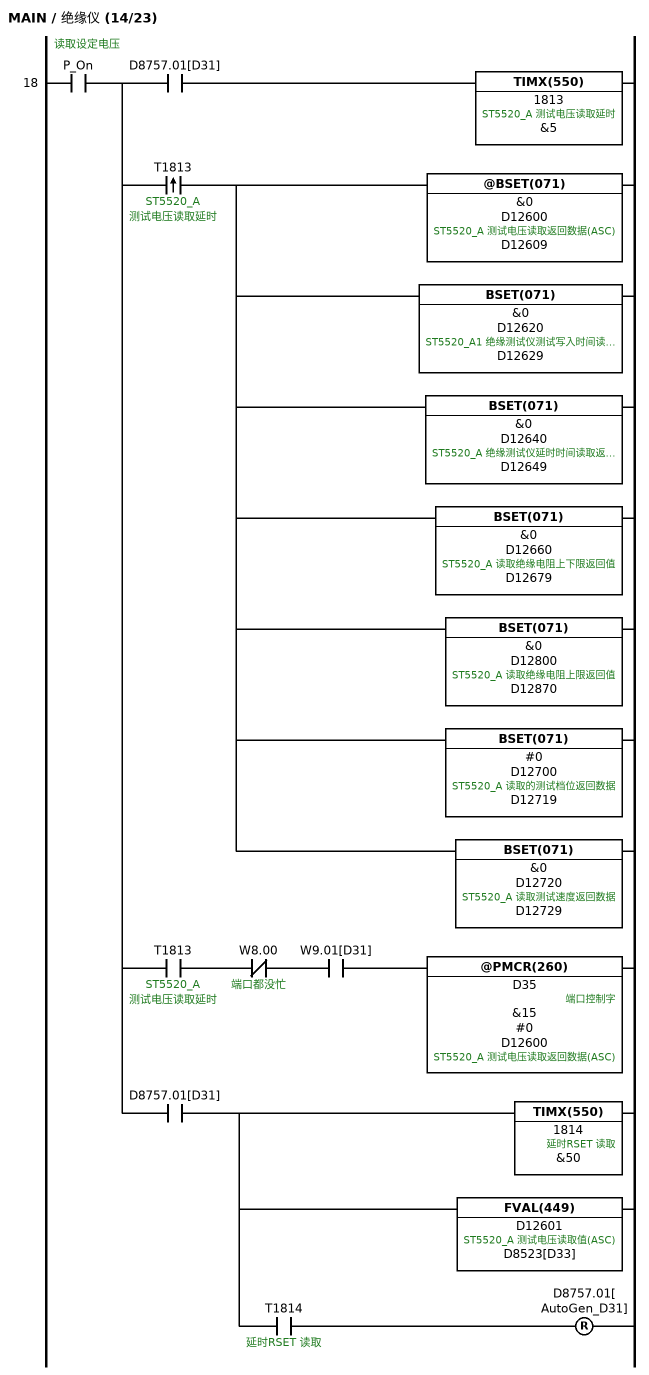
; [picture p48: MAIN / 绝缘仪, rungs 18-18]
; rung 18: 读取设定电压
LD P_On
OUT TR0
AND D8757.01[D31]
TIMX(550) 1813 &5  ; ST5520_A 测试电压读取延时
LD TR0
@AND T1813  ; ST5520_A 测试电压读取延时
@BSET(071) &0 D12600 D12609  ; ST5520_A 测试电压读取返回数据(ASC)
BSET(071) &0 D12620 D12629  ; ST5520_A1 绝缘测试仪测试写入时间读取值(ASC)
BSET(071) &0 D12640 D12649  ; ST5520_A 绝缘测试仪延时时间读取返回数据(ASC)
BSET(071) &0 D12660 D12679  ; ST5520_A 读取绝缘电阻上下限返回值
BSET(071) &0 D12800 D12870  ; ST5520_A 读取绝缘电阻上限返回值
BSET(071) #0 D12700 D12719  ; ST5520_A 读取的测试档位返回数据
BSET(071) &0 D12720 D12729  ; ST5520_A 读取测试速度返回数据
LD TR0
AND T1813  ; ST5520_A 测试电压读取延时
ANDNOT W8.00  ; 端口都没忙
AND W9.01[D31]
@PMCR(260) D35 &15 #0 D12600  ; 端口控制字, ST5520_A 测试电压读取返回数据(ASC)
LD TR0
AND D8757.01[D31]
TIMX(550) 1814 &50  ; 延时RSET 读取
FVAL(449) D12601 D8523[D33]  ; ST5520_A 测试电压读取值(ASC)
AND T1814  ; 延时RSET 读取
RSET D8757.01[AutoGen_D31]

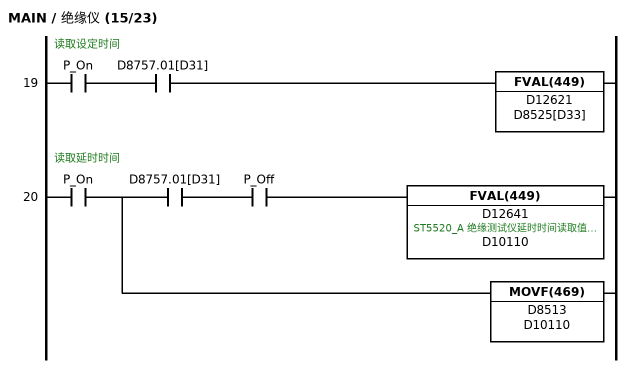
; rung 19: 读取设定时间
LD P_On
AND D8757.01[D31]
FVAL(449) D12621 D8525[D33]
; rung 20: 读取延时时间
LD P_On
OUT TR0
AND D8757.01[D31]
AND P_Off
FVAL(449) D12641 D10110  ; ST5520_A 绝缘测试仪延时时间读取值(ASC)
LD TR0
MOVF(469) D8513 D10110

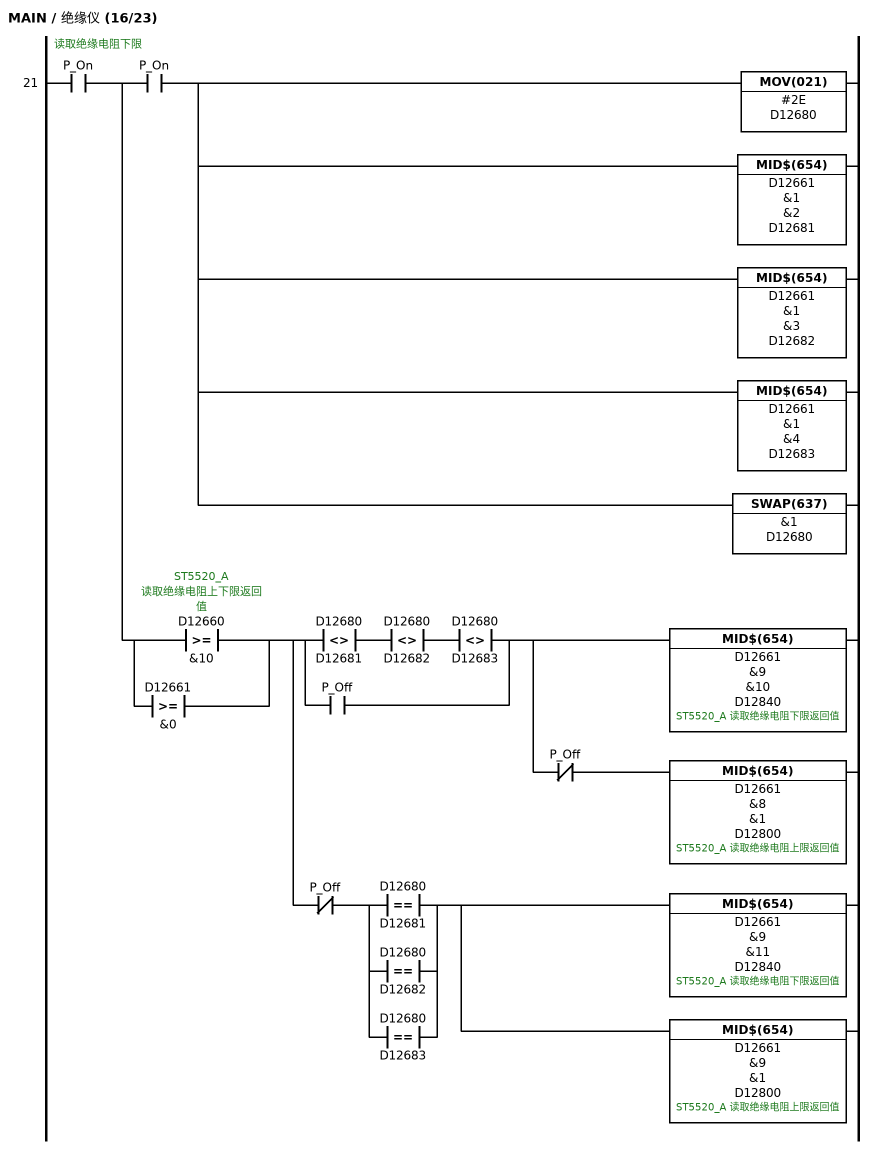
; rung 21: 读取绝缘电阻下限
LD P_On
OUT TR0
AND P_On
MOV(021) #2E D12680
MID$(654) D12661 &1 &2 D12681
MID$(654) D12661 &1 &3 D12682
MID$(654) D12661 &1 &4 D12683
SWAP(637) &1 D12680
LD TR0
LD>=(325) D12660 &10  ; ST5520_A 读取绝缘电阻上下限返回值
OR>=(325) D12661 &0
ANDLD
OUT TR0
LD<>(305) D12680 D12681
AND<>(305) D12680 D12682
AND<>(305) D12680 D12683
OR P_Off
ANDLD
MID$(654) D12661 &9 &10 D12840  ; ST5520_A 读取绝缘电阻下限返回值
ANDNOT P_Off
MID$(654) D12661 &8 &1 D12800  ; ST5520_A 读取绝缘电阻上限返回值
LD TR0
ANDNOT P_Off
LD=(300) D12680 D12681
OR=(300) D12680 D12682
OR=(300) D12680 D12683
ANDLD
MID$(654) D12661 &9 &11 D12840  ; ST5520_A 读取绝缘电阻下限返回值
MID$(654) D12661 &9 &1 D12800  ; ST5520_A 读取绝缘电阻上限返回值

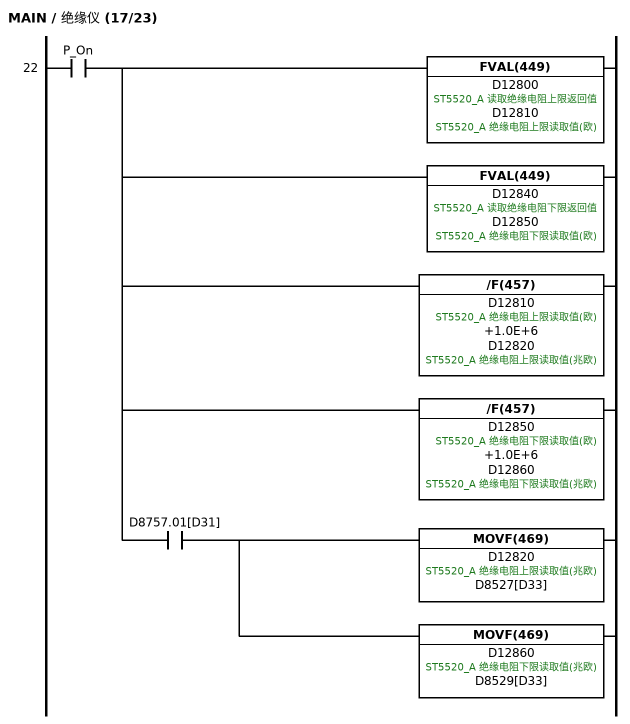
; rung 22
LD P_On
FVAL(449) D12800 D12810  ; ST5520_A 读取绝缘电阻上限返回值, ST5520_A 绝缘电阻上限读取值(欧)
FVAL(449) D12840 D12850  ; ST5520_A 读取绝缘电阻下限返回值, ST5520_A 绝缘电阻下限读取值(欧)
/F(457) D12810 +1.0E+6 D12820  ; ST5520_A 绝缘电阻上限读取值(欧), ST5520_A 绝缘电阻上限读取值(兆欧)
/F(457) D12850 +1.0E+6 D12860  ; ST5520_A 绝缘电阻下限读取值(欧), ST5520_A 绝缘电阻下限读取值(兆欧)
AND D8757.01[D31]
MOVF(469) D12820 D8527[D33]  ; ST5520_A 绝缘电阻上限读取值(兆欧)
MOVF(469) D12860 D8529[D33]  ; ST5520_A 绝缘电阻下限读取值(兆欧)

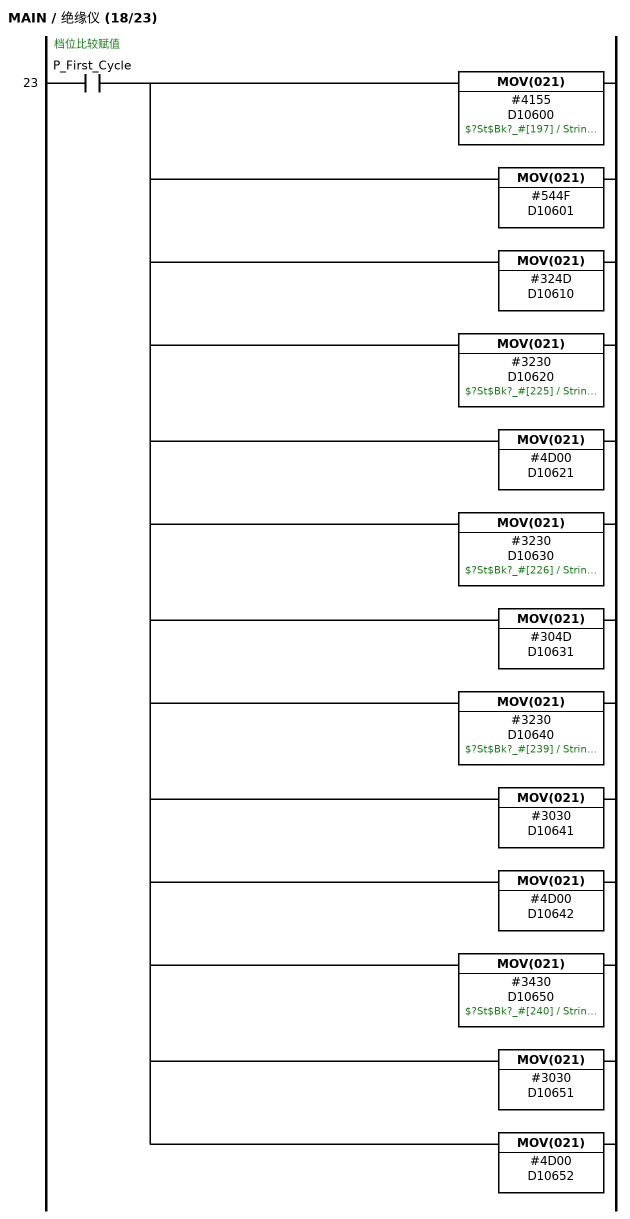
; rung 23: 档位比较赋值
LD P_First_Cycle
MOV(021) #4155 D10600  ; $?St$Bk?_#[197] / String "AUTO"$?St$Bk?_#[197]
MOV(021) #544F D10601
MOV(021) #324D D10610
MOV(021) #3230 D10620  ; $?St$Bk?_#[225] / String "20M"$?St$Bk?_#[225]
MOV(021) #4D00 D10621
MOV(021) #3230 D10630  ; $?St$Bk?_#[226] / String "200M"$?St$Bk?_#[226]
MOV(021) #304D D10631
MOV(021) #3230 D10640  ; $?St$Bk?_#[239] / String "2000M"$?St$Bk?_#[239]
MOV(021) #3030 D10641
MOV(021) #4D00 D10642
MOV(021) #3430 D10650  ; $?St$Bk?_#[240] / String "4000M"$?St$Bk?_#[240]
MOV(021) #3030 D10651
MOV(021) #4D00 D10652

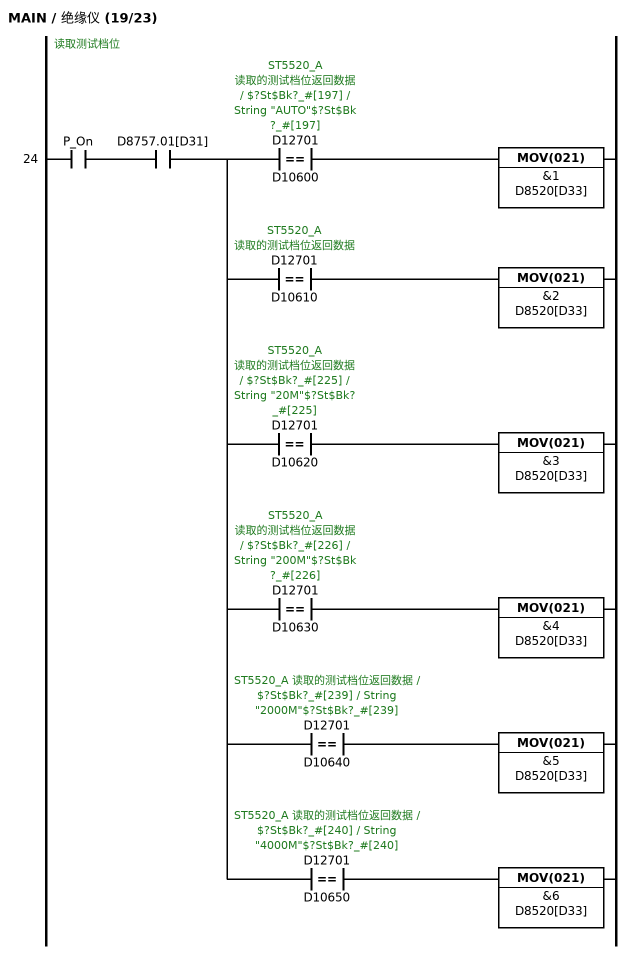
; rung 24: 读取测试档位
LD P_On
AND D8757.01[D31]
OUT TR0
AND=$(670) D12701 D10600  ; ST5520_A 读取的测试档位返回数据, $?St$Bk?_#[197] / String "AUTO"$?St$Bk?_#[197]
MOV(021) &1 D8520[D33]
LD TR0
AND=$(670) D12701 D10610  ; ST5520_A 读取的测试档位返回数据
MOV(021) &2 D8520[D33]
LD TR0
AND=$(670) D12701 D10620  ; ST5520_A 读取的测试档位返回数据, $?St$Bk?_#[225] / String "20M"$?St$Bk?_#[225]
MOV(021) &3 D8520[D33]
LD TR0
AND=$(670) D12701 D10630  ; ST5520_A 读取的测试档位返回数据, $?St$Bk?_#[226] / String "200M"$?St$Bk?_#[226]
MOV(021) &4 D8520[D33]
LD TR0
AND=$(670) D12701 D10640  ; ST5520_A 读取的测试档位返回数据, $?St$Bk?_#[239] / String "2000M"$?St$Bk?_#[239]
MOV(021) &5 D8520[D33]
LD TR0
AND=$(670) D12701 D10650  ; ST5520_A 读取的测试档位返回数据, $?St$Bk?_#[240] / String "4000M"$?St$Bk?_#[240]
MOV(021) &6 D8520[D33]

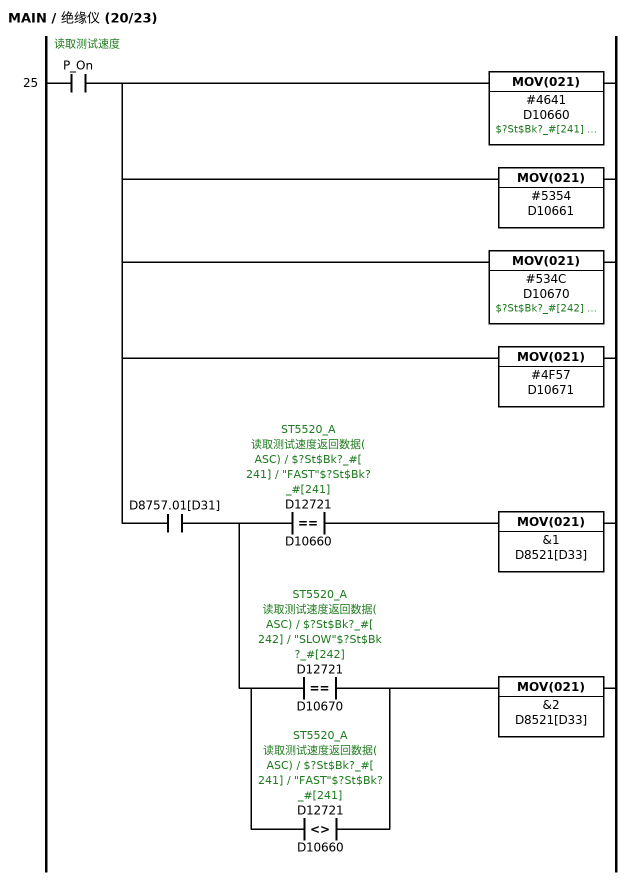
; rung 25: 读取测试速度
LD P_On
MOV(021) #4641 D10660  ; $?St$Bk?_#[241] / "FAST"$?St$Bk?_#[241]
MOV(021) #5354 D10661
MOV(021) #534C D10670  ; $?St$Bk?_#[242] / "SLOW"$?St$Bk?_#[242]
MOV(021) #4F57 D10671
AND D8757.01[D31]
OUT TR0
AND=$(670) D12721 D10660  ; ST5520_A 读取测试速度返回数据(ASC), $?St$Bk?_#[241] / "FAST"$?St$Bk?_#[241]
MOV(021) &1 D8521[D33]
LD TR0
LD=$(670) D12721 D10670  ; ST5520_A 读取测试速度返回数据(ASC), $?St$Bk?_#[242] / "SLOW"$?St$Bk?_#[242]
OR<>$(671) D12721 D10660  ; ST5520_A 读取测试速度返回数据(ASC), $?St$Bk?_#[241] / "FAST"$?St$Bk?_#[241]
ANDLD
MOV(021) &2 D8521[D33]

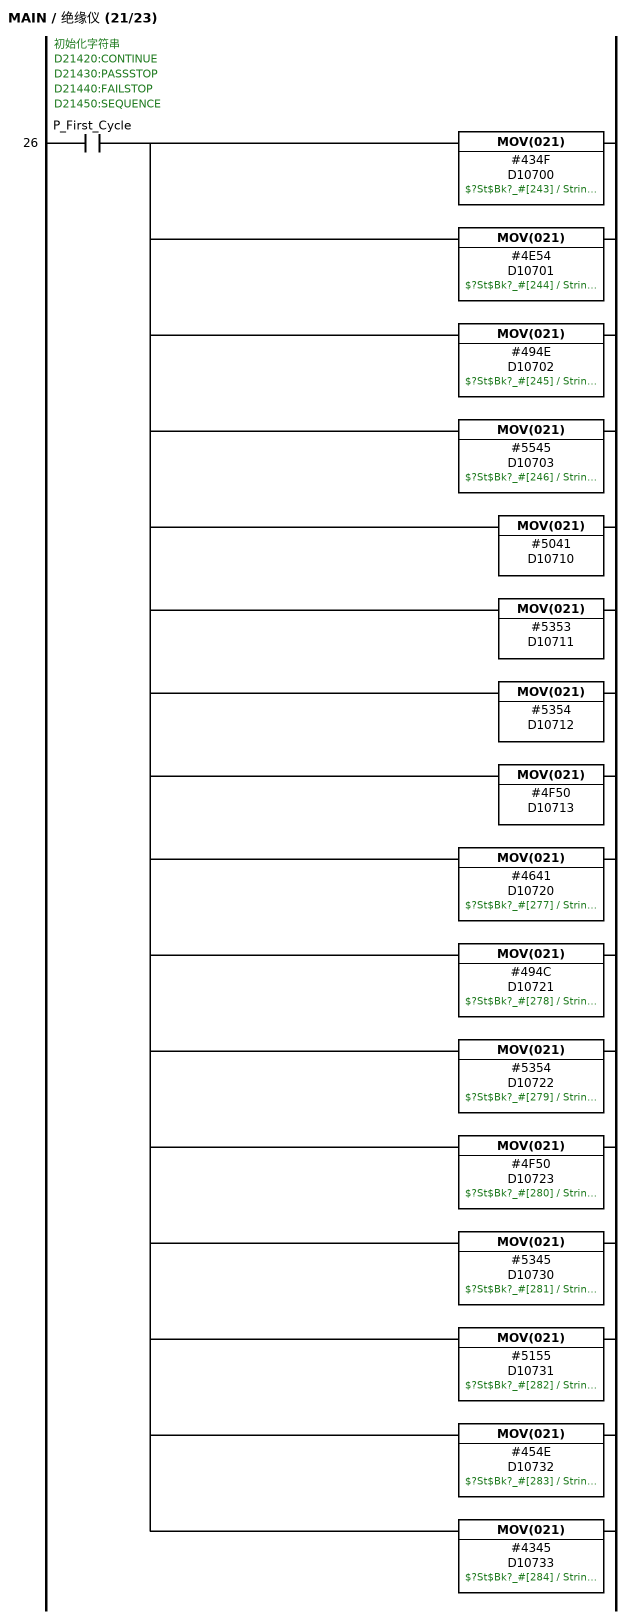
; rung 26: 初始化字符串 / D21420:CONTINUE / D21430:PASSSTOP / D21440:FAILSTOP / D21450:SEQUENCE
LD P_First_Cycle
MOV(021) #434F D10700  ; $?St$Bk?_#[243] / String "CONTINUE"$?St$Bk?_#[243]
MOV(021) #4E54 D10701  ; $?St$Bk?_#[244] / String "CONTINUE"$?St$Bk?_#[244]
MOV(021) #494E D10702  ; $?St$Bk?_#[245] / String "CONTINUE"$?St$Bk?_#[245]
MOV(021) #5545 D10703  ; $?St$Bk?_#[246] / String "CONTINUE"$?St$Bk?_#[246]
MOV(021) #5041 D10710
MOV(021) #5353 D10711
MOV(021) #5354 D10712
MOV(021) #4F50 D10713
MOV(021) #4641 D10720  ; $?St$Bk?_#[277] / String "FAILSTOP"$?St$Bk?_#[277]
MOV(021) #494C D10721  ; $?St$Bk?_#[278] / String "FAILSTOP"$?St$Bk?_#[278]
MOV(021) #5354 D10722  ; $?St$Bk?_#[279] / String "FAILSTOP"$?St$Bk?_#[279]
MOV(021) #4F50 D10723  ; $?St$Bk?_#[280] / String "FAILSTOP"$?St$Bk?_#[280]
MOV(021) #5345 D10730  ; $?St$Bk?_#[281] / String "SEQUENCE"$?St$Bk?_#[281]
MOV(021) #5155 D10731  ; $?St$Bk?_#[282] / String "SEQUENCE"$?St$Bk?_#[282]
MOV(021) #454E D10732  ; $?St$Bk?_#[283] / String "SEQUENCE"$?St$Bk?_#[283]
MOV(021) #4345 D10733  ; $?St$Bk?_#[284] / String "SEQUENCE"$?St$Bk?_#[284]

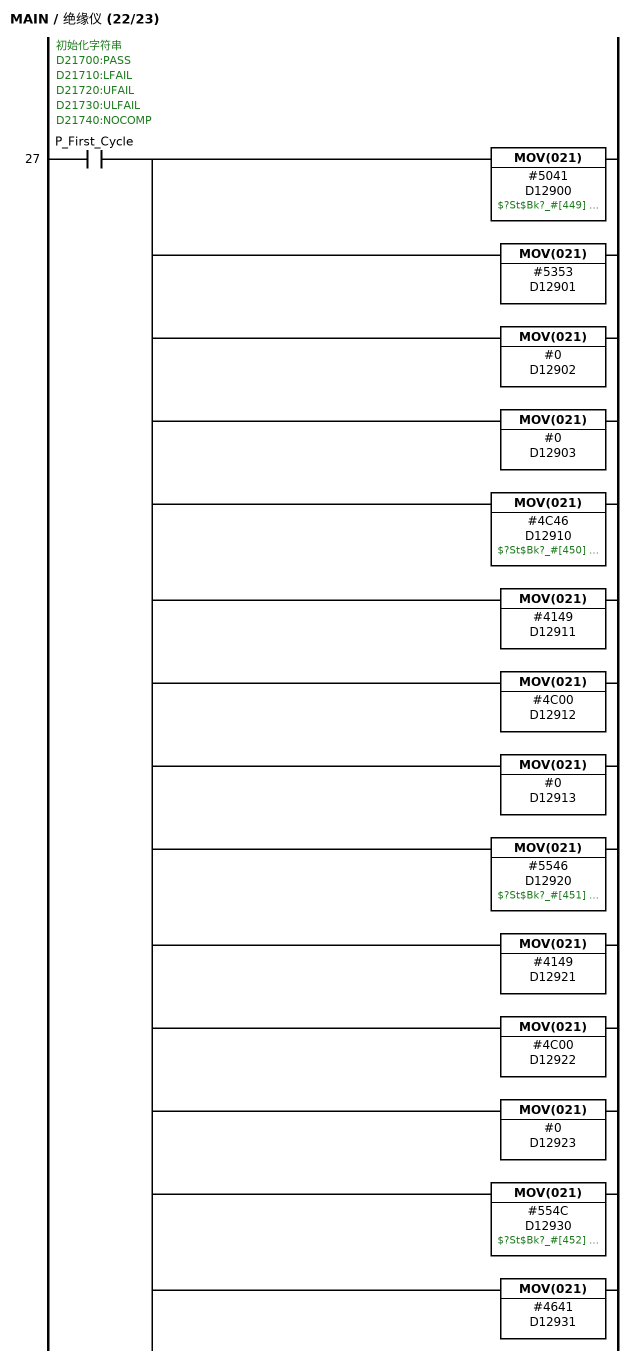

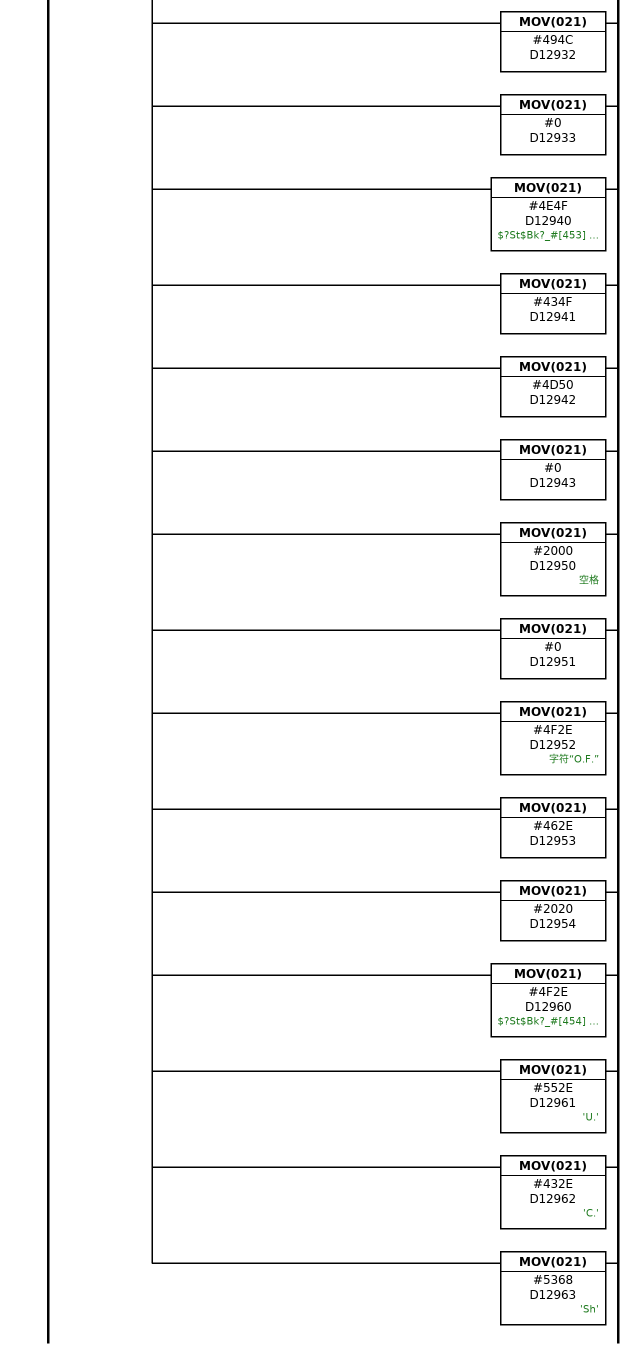
; rung 27: 初始化字符串 / D21700:PASS / D21710:LFAIL / D21720:UFAIL / D21730:ULFAIL / D21740:NOCOMP
LD P_First_Cycle
MOV(021) #5041 D12900  ; $?St$Bk?_#[449] / "PASS"$?St$Bk?_#[449]
MOV(021) #5353 D12901
MOV(021) #0 D12902
MOV(021) #0 D12903
MOV(021) #4C46 D12910  ; $?St$Bk?_#[450] / "LFAIL"$?St$Bk?_#[450]
MOV(021) #4149 D12911
MOV(021) #4C00 D12912
MOV(021) #0 D12913
MOV(021) #5546 D12920  ; $?St$Bk?_#[451] / "UFAIL"$?St$Bk?_#[451]
MOV(021) #4149 D12921
MOV(021) #4C00 D12922
MOV(021) #0 D12923
MOV(021) #554C D12930  ; $?St$Bk?_#[452] / "ULFAIL"$?St$Bk?_#[452]
MOV(021) #4641 D12931
MOV(021) #494C D12932
MOV(021) #0 D12933
MOV(021) #4E4F D12940  ; $?St$Bk?_#[453] / "NOCOMP"$?St$Bk?_#[453]
MOV(021) #434F D12941
MOV(021) #4D50 D12942
MOV(021) #0 D12943
MOV(021) #2000 D12950  ; 空格
MOV(021) #0 D12951
MOV(021) #4F2E D12952  ; 字符“O.F.”
MOV(021) #462E D12953
MOV(021) #2020 D12954
MOV(021) #4F2E D12960  ; $?St$Bk?_#[454] / "O."$?St$Bk?_#[454]
MOV(021) #552E D12961  ; 'U.'
MOV(021) #432E D12962  ; 'C.'
MOV(021) #5368 D12963  ; 'Sh'

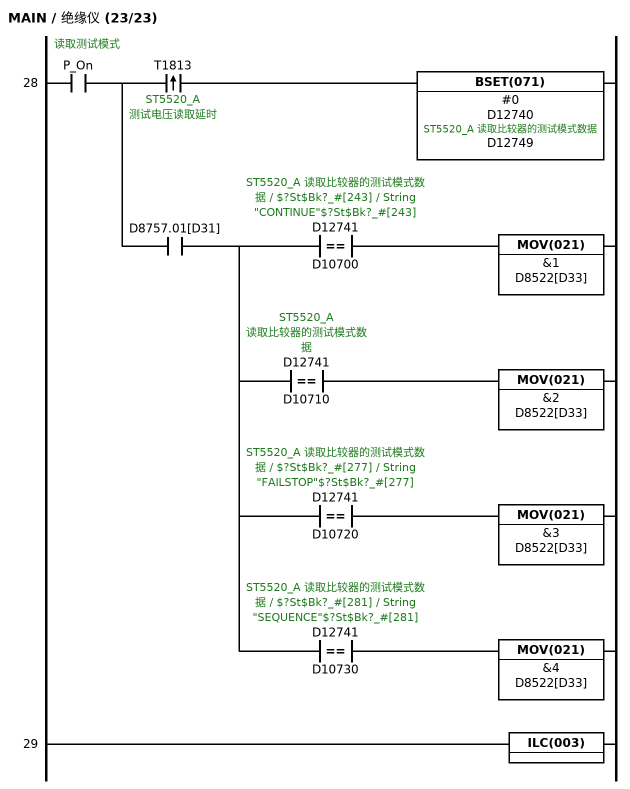
; rung 28: 读取测试模式
LD P_On
OUT TR0
@AND T1813  ; ST5520_A 测试电压读取延时
BSET(071) #0 D12740 D12749  ; ST5520_A 读取比较器的测试模式数据
LD TR0
AND D8757.01[D31]
OUT TR0
AND=$(670) D12741 D10700  ; ST5520_A 读取比较器的测试模式数据, $?St$Bk?_#[243] / String "CONTINUE"$?St$Bk?_#[243]
MOV(021) &1 D8522[D33]
LD TR0
AND=$(670) D12741 D10710  ; ST5520_A 读取比较器的测试模式数据
MOV(021) &2 D8522[D33]
LD TR0
AND=$(670) D12741 D10720  ; ST5520_A 读取比较器的测试模式数据, $?St$Bk?_#[277] / String "FAILSTOP"$?St$Bk?_#[277]
MOV(021) &3 D8522[D33]
LD TR0
AND=$(670) D12741 D10730  ; ST5520_A 读取比较器的测试模式数据, $?St$Bk?_#[281] / String "SEQUENCE"$?St$Bk?_#[281]
MOV(021) &4 D8522[D33]
; rung 29
ILC(003)

### Section 测试自动

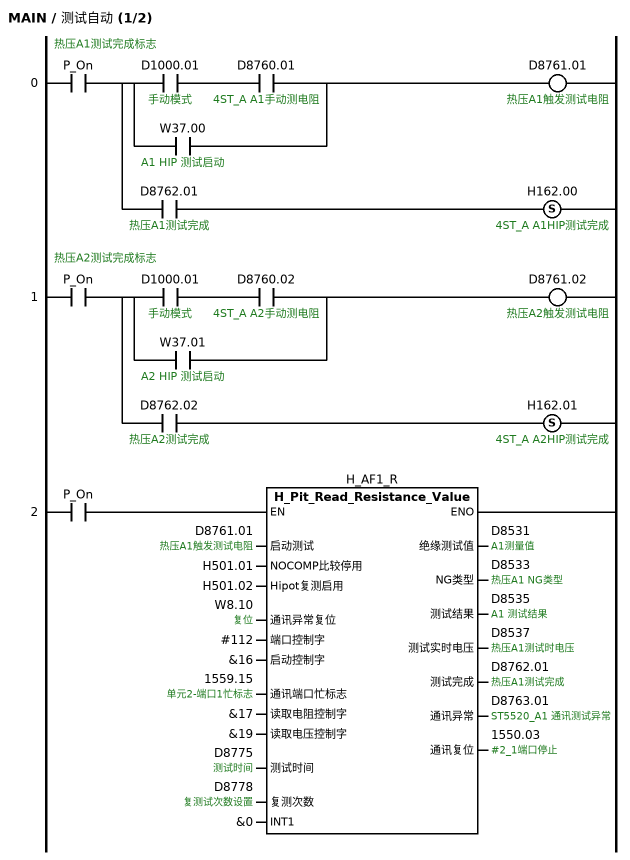
; rung 0: 热压A1测试完成标志
LD P_On
OUT TR0
LD D1000.01  ; 手动模式
AND D8760.01  ; 4ST_A A1手动测电阻
OR W37.00  ; A1 HIP 测试启动
ANDLD
OUT D8761.01  ; 热压A1触发测试电阻
LD TR0
AND D8762.01  ; 热压A1测试完成
SET H162.00  ; 4ST_A A1HIP测试完成
; rung 1: 热压A2测试完成标志
LD P_On
OUT TR0
LD D1000.01  ; 手动模式
AND D8760.02  ; 4ST_A A2手动测电阻
OR W37.01  ; A2 HIP 测试启动
ANDLD
OUT D8761.02  ; 热压A2触发测试电阻
LD TR0
AND D8762.02  ; 热压A2测试完成
SET H162.01  ; 4ST_A A2HIP测试完成
; rung 2
LD P_On
CALL H_AF1_R : H_Pit_Read_Resistance_Value (启动测试 := D8761.01, NOCOMP比较停用 := H501.01, Hipot复测启用 := H501.02, 通讯异常复位 := W8.10, 端口控制字 := #112, 启动控制字 := &16, 通讯端口忙标志 := 1559.15, 读取电阻控制字 := &17, 读取电压控制字 := &19, 测试时间 := D8775, 复测次数 := D8778, INT1 := &0, 绝缘测试值 => D8531, NG类型 => D8533, 测试结果 => D8535, 测试实时电压 => D8537, 测试完成 => D8762.01, 通讯异常 => D8763.01, 通讯复位 => 1550.03)  ; 热压A1触发测试电阻, 复位, 单元2-端口1忙标志, 测试时间, 复测试次数设置, A1测量值, 热压A1 NG类型, A1 测试结果, 热压A1测试时电压, 热压A1测试完成, ST5520_A1 通讯测试异常, #2_1端口停止

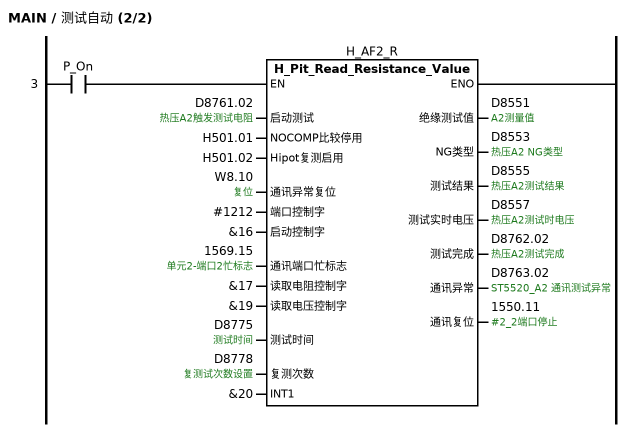
; rung 3
LD P_On
CALL H_AF2_R : H_Pit_Read_Resistance_Value (启动测试 := D8761.02, NOCOMP比较停用 := H501.01, Hipot复测启用 := H501.02, 通讯异常复位 := W8.10, 端口控制字 := #1212, 启动控制字 := &16, 通讯端口忙标志 := 1569.15, 读取电阻控制字 := &17, 读取电压控制字 := &19, 测试时间 := D8775, 复测次数 := D8778, INT1 := &20, 绝缘测试值 => D8551, NG类型 => D8553, 测试结果 => D8555, 测试实时电压 => D8557, 测试完成 => D8762.02, 通讯异常 => D8763.02, 通讯复位 => 1550.11)  ; 热压A2触发测试电阻, 复位, 单元2-端口2忙标志, 测试时间, 复测试次数设置, A2测量值, 热压A2 NG类型, 热压A2测试结果, 热压A2测试时电压, 热压A2测试完成, ST5520_A2 通讯测试异常, #2_2端口停止

### Section END
; rung 0
END(001)

## Program 进料定位 (cyclic task 1)

### Section Main

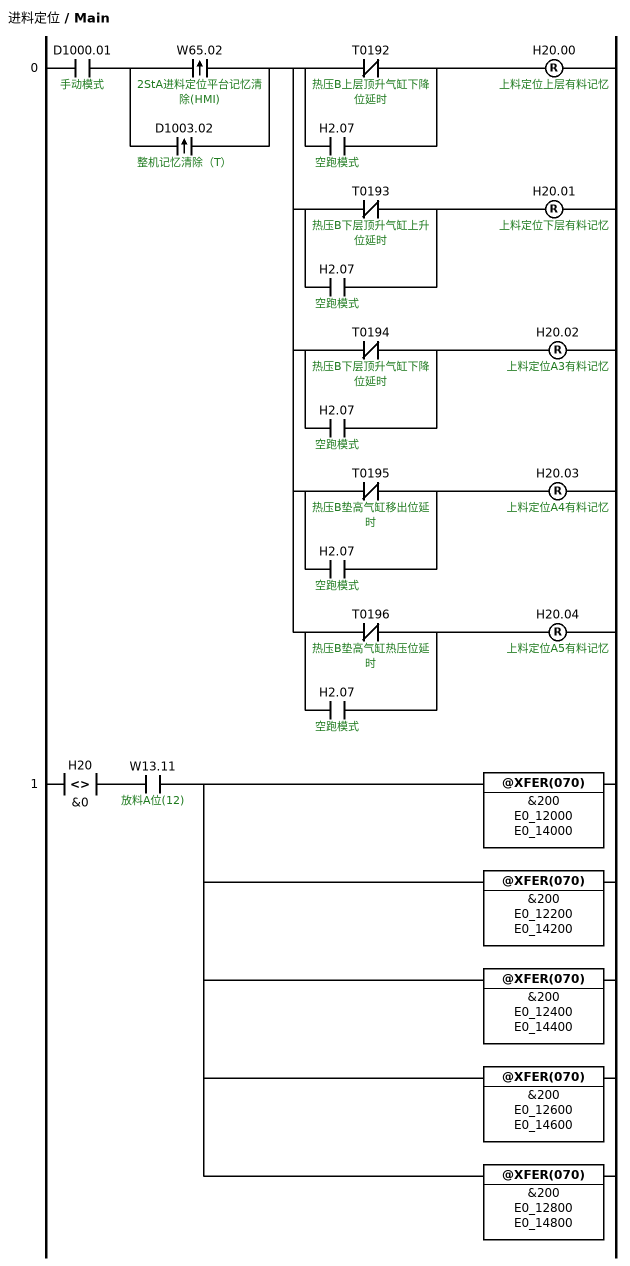
; rung 0
LD D1000.01  ; 手动模式
@LD W65.02  ; 2StA进料定位平台记忆清除(HMI)
@OR D1003.02  ; 整机记忆清除（T）
ANDLD
OUT TR0
LDNOT T0192  ; 热压B上层顶升气缸下降位延时
OR H2.07  ; 空跑模式
ANDLD
RSET H20.00  ; 上料定位上层有料记忆
LD TR0
LDNOT T0193  ; 热压B下层顶升气缸上升位延时
OR H2.07  ; 空跑模式
ANDLD
RSET H20.01  ; 上料定位下层有料记忆
LD TR0
LDNOT T0194  ; 热压B下层顶升气缸下降位延时
OR H2.07  ; 空跑模式
ANDLD
RSET H20.02  ; 上料定位A3有料记忆
LD TR0
LDNOT T0195  ; 热压B垫高气缸移出位延时
OR H2.07  ; 空跑模式
ANDLD
RSET H20.03  ; 上料定位A4有料记忆
LD TR0
LDNOT T0196  ; 热压B垫高气缸热压位延时
OR H2.07  ; 空跑模式
ANDLD
RSET H20.04  ; 上料定位A5有料记忆
; rung 1
LD<>(305) H20 &0
AND W13.11  ; 放料A位(12)
@XFER(070) &200 E0_12000 E0_14000
@XFER(070) &200 E0_12200 E0_14200
@XFER(070) &200 E0_12400 E0_14400
@XFER(070) &200 E0_12600 E0_14600
@XFER(070) &200 E0_12800 E0_14800

### Section _1ST进料定位

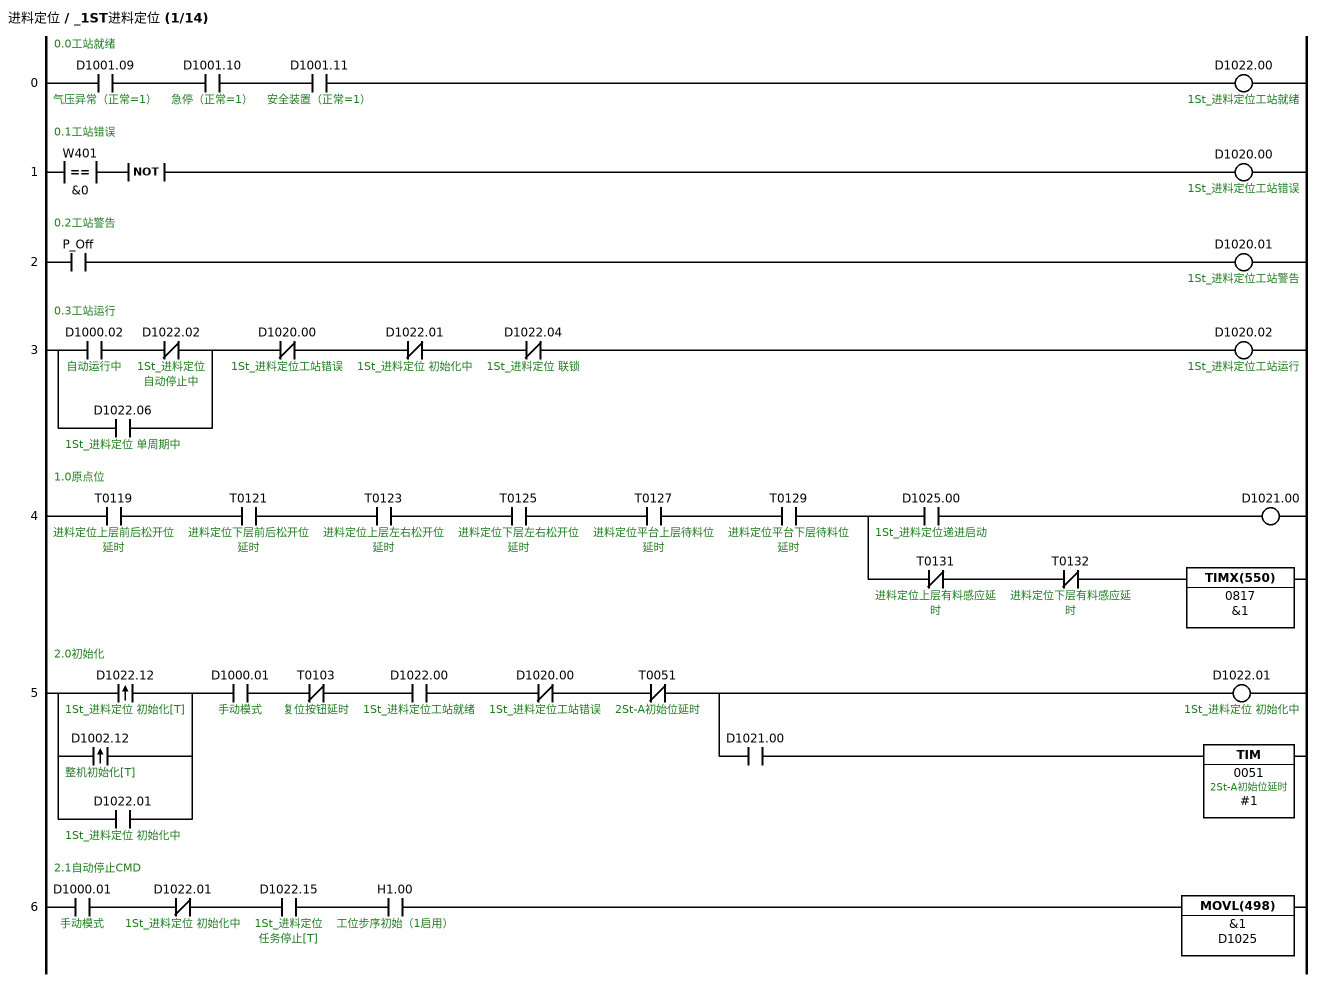
; rung 0: 0.0工站就绪
LD D1001.09  ; 气压异常（正常=1）
AND D1001.10  ; 急停（正常=1）
AND D1001.11  ; 安全装置（正常=1）
OUT D1022.00  ; 1St_进料定位工站就绪
; rung 1: 0.1工站错误
LD=(300) W401 &0
NOT(520)
OUT D1020.00  ; 1St_进料定位工站错误
; rung 2: 0.2工站警告
LD P_Off
OUT D1020.01  ; 1St_进料定位工站警告
; rung 3: 0.3工站运行
LD D1000.02  ; 自动运行中
ANDNOT D1022.02  ; 1St_进料定位 自动停止中
OR D1022.06  ; 1St_进料定位 单周期中
ANDNOT D1020.00  ; 1St_进料定位工站错误
ANDNOT D1022.01  ; 1St_进料定位 初始化中
ANDNOT D1022.04  ; 1St_进料定位 联锁
OUT D1020.02  ; 1St_进料定位工站运行
; rung 4: 1.0原点位
LD T0119  ; 进料定位上层前后松开位延时
AND T0121  ; 进料定位下层前后松开位延时
AND T0123  ; 进料定位上层左右松开位延时
AND T0125  ; 进料定位下层左右松开位延时
AND T0127  ; 进料定位平台上层待料位延时
AND T0129  ; 进料定位平台下层待料位延时
OUT TR0
AND D1025.00  ; 1St_进料定位递进启动
OUT D1021.00
LD TR0
ANDNOT T0131  ; 进料定位上层有料感应延时
ANDNOT T0132  ; 进料定位下层有料感应延时
TIMX(550) 0817 &1
; rung 5: 2.0初始化
@LD D1022.12  ; 1St_进料定位 初始化[T]
@OR D1002.12  ; 整机初始化[T]
OR D1022.01  ; 1St_进料定位 初始化中
AND D1000.01  ; 手动模式
ANDNOT T0103  ; 复位按钮延时
AND D1022.00  ; 1St_进料定位工站就绪
ANDNOT D1020.00  ; 1St_进料定位工站错误
ANDNOT T0051  ; 2St-A初始位延时
OUT D1022.01  ; 1St_进料定位 初始化中
AND D1021.00
TIM 0051 #1  ; 2St-A初始位延时
; rung 6: 2.1自动停止CMD
LD D1000.01  ; 手动模式
ANDNOT D1022.01  ; 1St_进料定位 初始化中
AND D1022.15  ; 1St_进料定位 任务停止[T]
AND H1.00  ; 工位步序初始（1启用）
MOVL(498) &1 D1025

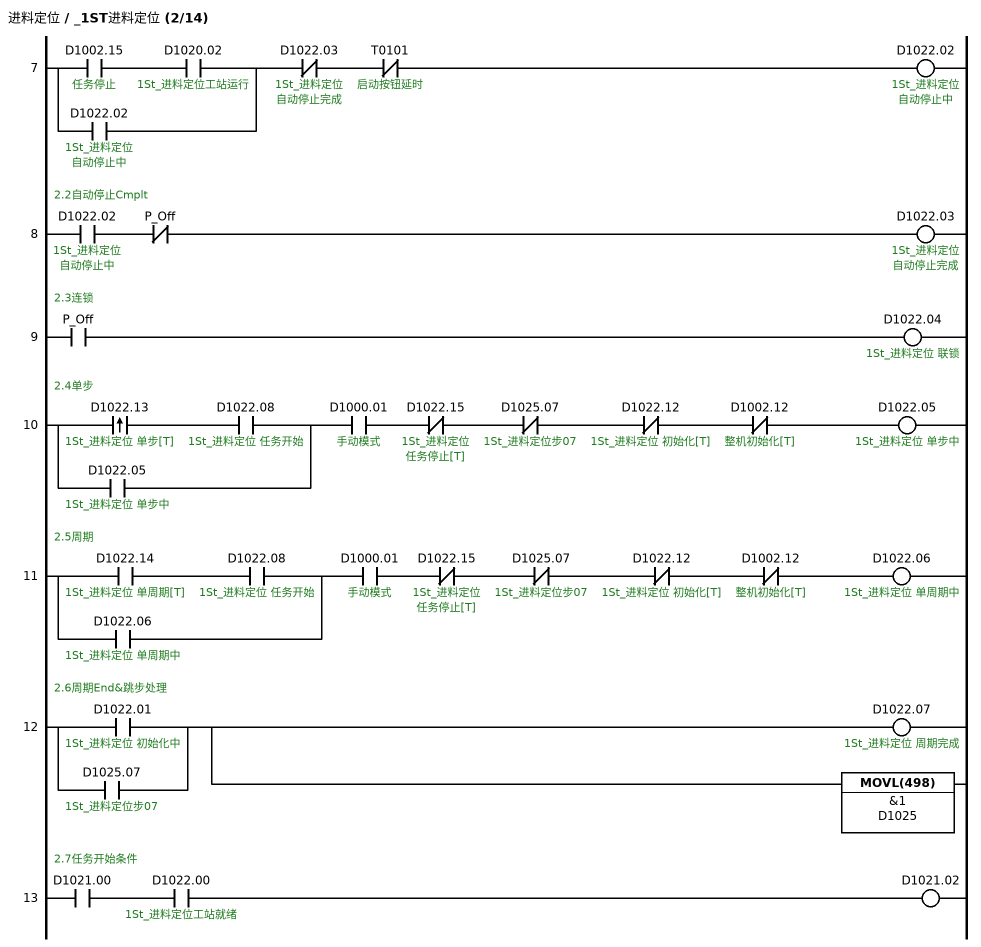
; rung 7
LD D1002.15  ; 任务停止
AND D1020.02  ; 1St_进料定位工站运行
OR D1022.02  ; 1St_进料定位 自动停止中
ANDNOT D1022.03  ; 1St_进料定位 自动停止完成
ANDNOT T0101  ; 启动按钮延时
OUT D1022.02  ; 1St_进料定位 自动停止中
; rung 8: 2.2自动停止Cmplt
LD D1022.02  ; 1St_进料定位 自动停止中
ANDNOT P_Off
OUT D1022.03  ; 1St_进料定位 自动停止完成
; rung 9: 2.3连锁
LD P_Off
OUT D1022.04  ; 1St_进料定位 联锁
; rung 10: 2.4单步
@LD D1022.13  ; 1St_进料定位 单步[T]
AND D1022.08  ; 1St_进料定位 任务开始
OR D1022.05  ; 1St_进料定位 单步中
AND D1000.01  ; 手动模式
ANDNOT D1022.15  ; 1St_进料定位 任务停止[T]
ANDNOT D1025.07  ; 1St_进料定位步07
ANDNOT D1022.12  ; 1St_进料定位 初始化[T]
ANDNOT D1002.12  ; 整机初始化[T]
OUT D1022.05  ; 1St_进料定位 单步中
; rung 11: 2.5周期
LD D1022.14  ; 1St_进料定位 单周期[T]
AND D1022.08  ; 1St_进料定位 任务开始
OR D1022.06  ; 1St_进料定位 单周期中
AND D1000.01  ; 手动模式
ANDNOT D1022.15  ; 1St_进料定位 任务停止[T]
ANDNOT D1025.07  ; 1St_进料定位步07
ANDNOT D1022.12  ; 1St_进料定位 初始化[T]
ANDNOT D1002.12  ; 整机初始化[T]
OUT D1022.06  ; 1St_进料定位 单周期中
; rung 12: 2.6周期End&跳步处理
LD D1022.01  ; 1St_进料定位 初始化中
OR D1025.07  ; 1St_进料定位步07
OUT D1022.07  ; 1St_进料定位 周期完成
MOVL(498) &1 D1025
; rung 13: 2.7任务开始条件
LD D1021.00
AND D1022.00  ; 1St_进料定位工站就绪
OUT D1021.02

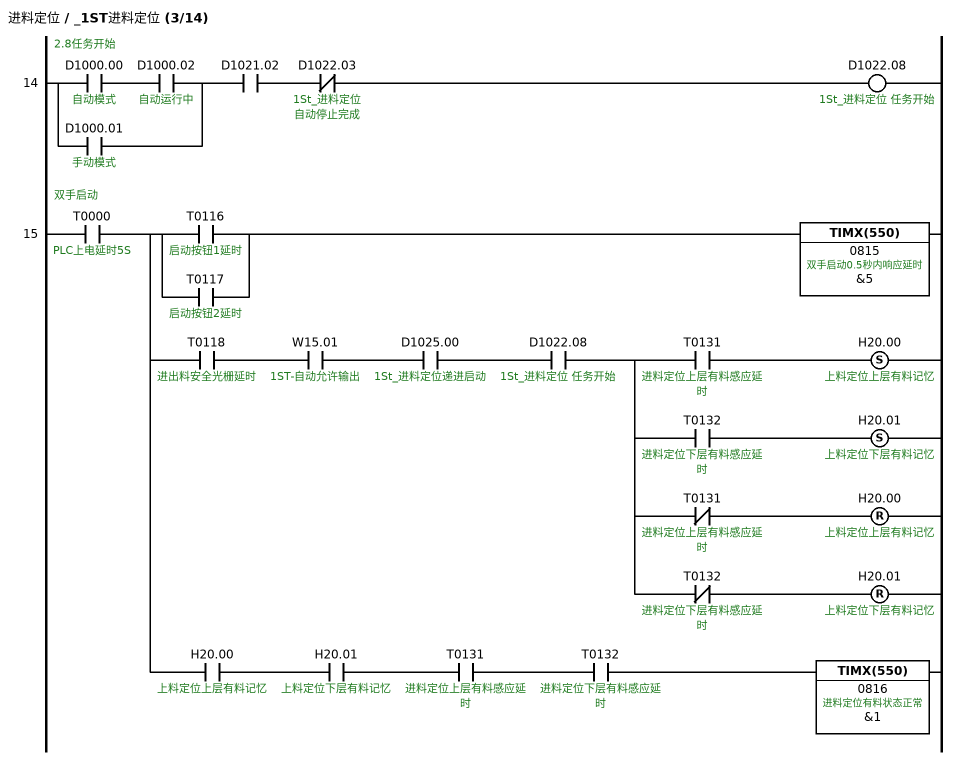
; rung 14: 2.8任务开始
LD D1000.00  ; 自动模式
AND D1000.02  ; 自动运行中
OR D1000.01  ; 手动模式
AND D1021.02
ANDNOT D1022.03  ; 1St_进料定位 自动停止完成
OUT D1022.08  ; 1St_进料定位 任务开始
; rung 15: 双手启动
LD T0000  ; PLC上电延时5S
OUT TR0
LD T0116  ; 启动按钮1延时
OR T0117  ; 启动按钮2延时
ANDLD
TIMX(550) 0815 &5  ; 双手启动0.5秒内响应延时
LD TR0
AND T0118  ; 进出料安全光栅延时
AND W15.01  ; 1ST-自动允许输出
AND D1025.00  ; 1St_进料定位递进启动
AND D1022.08  ; 1St_进料定位 任务开始
OUT TR1
AND T0131  ; 进料定位上层有料感应延时
SET H20.00  ; 上料定位上层有料记忆
LD TR1
AND T0132  ; 进料定位下层有料感应延时
SET H20.01  ; 上料定位下层有料记忆
LD TR1
ANDNOT T0131  ; 进料定位上层有料感应延时
RSET H20.00  ; 上料定位上层有料记忆
LD TR1
ANDNOT T0132  ; 进料定位下层有料感应延时
RSET H20.01  ; 上料定位下层有料记忆
LD TR0
AND H20.00  ; 上料定位上层有料记忆
AND H20.01  ; 上料定位下层有料记忆
AND T0131  ; 进料定位上层有料感应延时
AND T0132  ; 进料定位下层有料感应延时
TIMX(550) 0816 &1  ; 进料定位有料状态正常

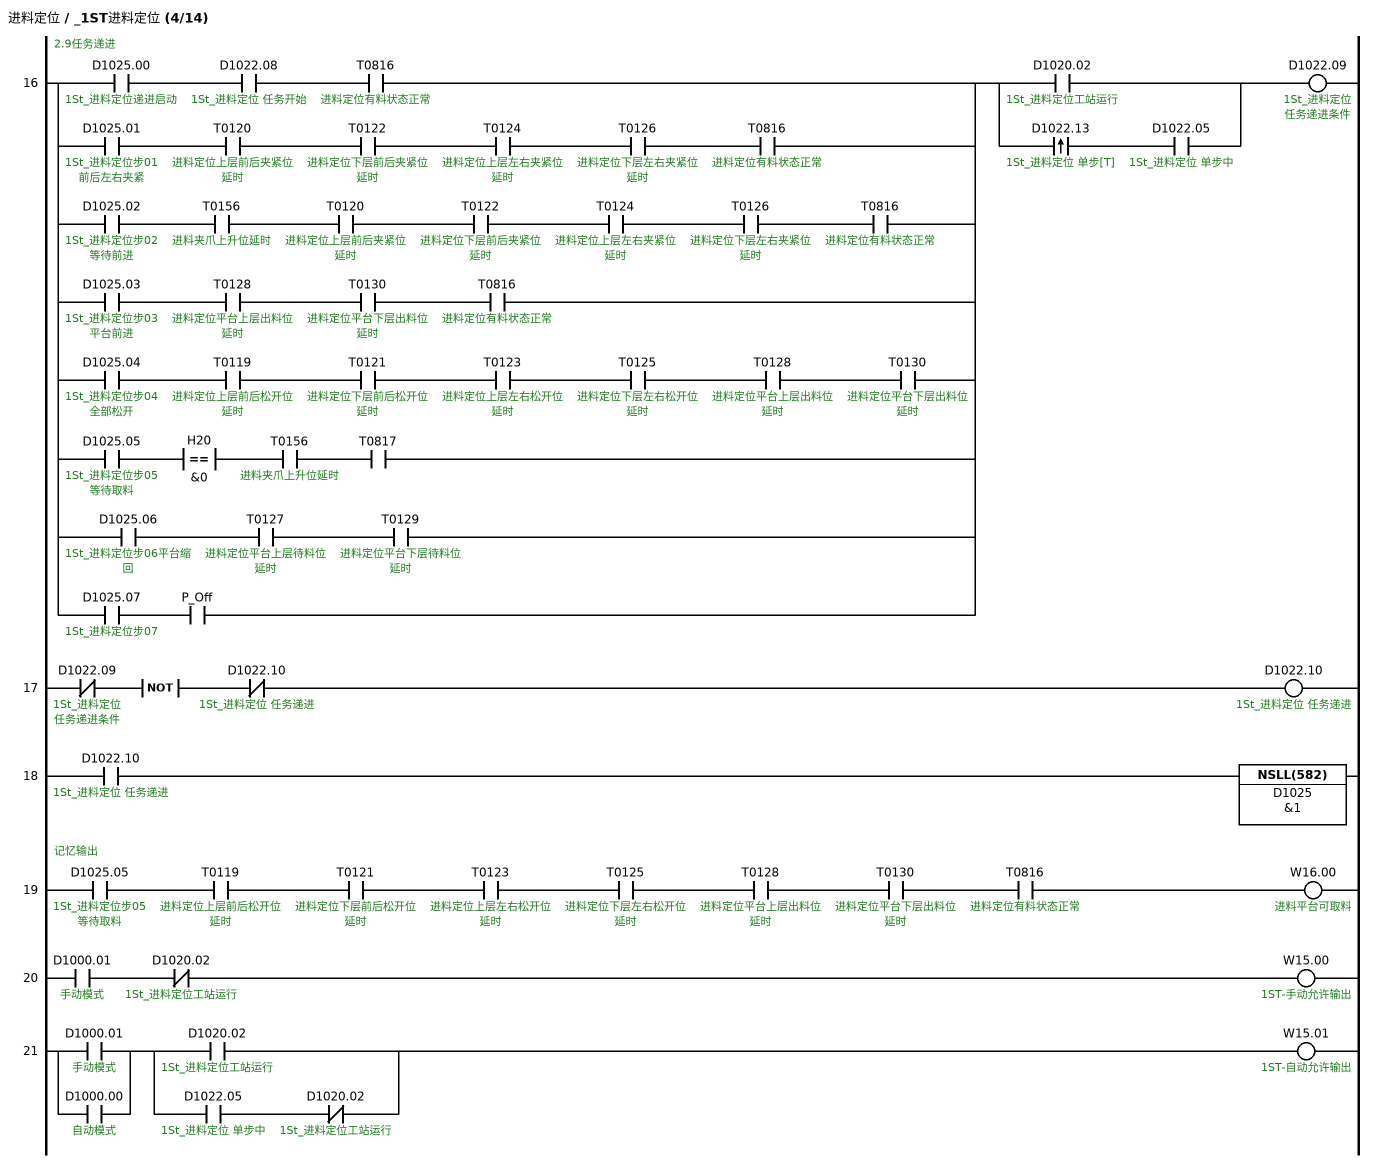
; rung 16: 2.9任务递进
LD D1025.00  ; 1St_进料定位递进启动
AND D1022.08  ; 1St_进料定位 任务开始
AND T0816  ; 进料定位有料状态正常
LD D1025.01  ; 1St_进料定位步01 前后左右夹紧
AND T0120  ; 进料定位上层前后夹紧位延时
AND T0122  ; 进料定位下层前后夹紧位延时
AND T0124  ; 进料定位上层左右夹紧位延时
AND T0126  ; 进料定位下层左右夹紧位延时
AND T0816  ; 进料定位有料状态正常
ORLD
LD D1025.02  ; 1St_进料定位步02 等待前进
AND T0156  ; 进料夹爪上升位延时
AND T0120  ; 进料定位上层前后夹紧位延时
AND T0122  ; 进料定位下层前后夹紧位延时
AND T0124  ; 进料定位上层左右夹紧位延时
AND T0126  ; 进料定位下层左右夹紧位延时
AND T0816  ; 进料定位有料状态正常
ORLD
LD D1025.03  ; 1St_进料定位步03 平台前进
AND T0128  ; 进料定位平台上层出料位延时
AND T0130  ; 进料定位平台下层出料位延时
AND T0816  ; 进料定位有料状态正常
ORLD
LD D1025.04  ; 1St_进料定位步04 全部松开
AND T0119  ; 进料定位上层前后松开位延时
AND T0121  ; 进料定位下层前后松开位延时
AND T0123  ; 进料定位上层左右松开位延时
AND T0125  ; 进料定位下层左右松开位延时
AND T0128  ; 进料定位平台上层出料位延时
AND T0130  ; 进料定位平台下层出料位延时
ORLD
LD D1025.05  ; 1St_进料定位步05 等待取料
AND=(300) H20 &0
AND T0156  ; 进料夹爪上升位延时
AND T0817
ORLD
LD D1025.06  ; 1St_进料定位步06平台缩回
AND T0127  ; 进料定位平台上层待料位延时
AND T0129  ; 进料定位平台下层待料位延时
ORLD
LD D1025.07  ; 1St_进料定位步07
AND P_Off
ORLD
LD D1020.02  ; 1St_进料定位工站运行
@LD D1022.13  ; 1St_进料定位 单步[T]
AND D1022.05  ; 1St_进料定位 单步中
ORLD
ANDLD
OUT D1022.09  ; 1St_进料定位 任务递进条件
; rung 17
LDNOT D1022.09  ; 1St_进料定位 任务递进条件
NOT(520)
ANDNOT D1022.10  ; 1St_进料定位 任务递进
OUT D1022.10  ; 1St_进料定位 任务递进
; rung 18
LD D1022.10  ; 1St_进料定位 任务递进
NSLL(582) D1025 &1
; rung 19: 记忆输出
LD D1025.05  ; 1St_进料定位步05 等待取料
AND T0119  ; 进料定位上层前后松开位延时
AND T0121  ; 进料定位下层前后松开位延时
AND T0123  ; 进料定位上层左右松开位延时
AND T0125  ; 进料定位下层左右松开位延时
AND T0128  ; 进料定位平台上层出料位延时
AND T0130  ; 进料定位平台下层出料位延时
AND T0816  ; 进料定位有料状态正常
OUT W16.00  ; 进料平台可取料
; rung 20
LD D1000.01  ; 手动模式
ANDNOT D1020.02  ; 1St_进料定位工站运行
OUT W15.00  ; 1ST-手动允许输出
; rung 21
LD D1000.01  ; 手动模式
OR D1000.00  ; 自动模式
LD D1020.02  ; 1St_进料定位工站运行
LD D1022.05  ; 1St_进料定位 单步中
ANDNOT D1020.02  ; 1St_进料定位工站运行
ORLD
ANDLD
OUT W15.01  ; 1ST-自动允许输出

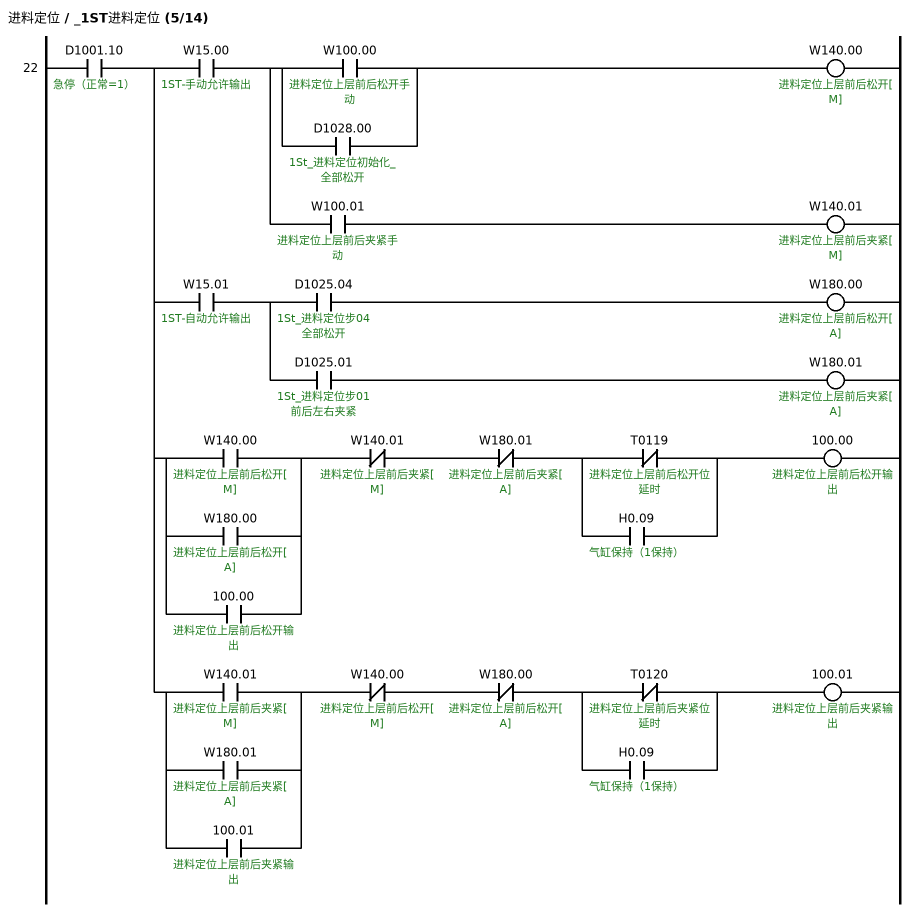
; rung 22
LD D1001.10  ; 急停（正常=1）
OUT TR0
AND W15.00  ; 1ST-手动允许输出
OUT TR1
LD W100.00  ; 进料定位上层前后松开手动
OR D1028.00  ; 1St_进料定位初始化_全部松开
ANDLD
OUT W140.00  ; 进料定位上层前后松开[M]
LD TR1
AND W100.01  ; 进料定位上层前后夹紧手动
OUT W140.01  ; 进料定位上层前后夹紧[M]
LD TR0
AND W15.01  ; 1ST-自动允许输出
OUT TR1
AND D1025.04  ; 1St_进料定位步04 全部松开
OUT W180.00  ; 进料定位上层前后松开[A]
LD TR1
AND D1025.01  ; 1St_进料定位步01 前后左右夹紧
OUT W180.01  ; 进料定位上层前后夹紧[A]
LD TR0
LD W140.00  ; 进料定位上层前后松开[M]
OR W180.00  ; 进料定位上层前后松开[A]
OR 100.00  ; 进料定位上层前后松开输出
ANDLD
ANDNOT W140.01  ; 进料定位上层前后夹紧[M]
ANDNOT W180.01  ; 进料定位上层前后夹紧[A]
LDNOT T0119  ; 进料定位上层前后松开位延时
OR H0.09  ; 气缸保持（1保持）
ANDLD
OUT 100.00  ; 进料定位上层前后松开输出
LD TR0
LD W140.01  ; 进料定位上层前后夹紧[M]
OR W180.01  ; 进料定位上层前后夹紧[A]
OR 100.01  ; 进料定位上层前后夹紧输出
ANDLD
ANDNOT W140.00  ; 进料定位上层前后松开[M]
ANDNOT W180.00  ; 进料定位上层前后松开[A]
LDNOT T0120  ; 进料定位上层前后夹紧位延时
OR H0.09  ; 气缸保持（1保持）
ANDLD
OUT 100.01  ; 进料定位上层前后夹紧输出

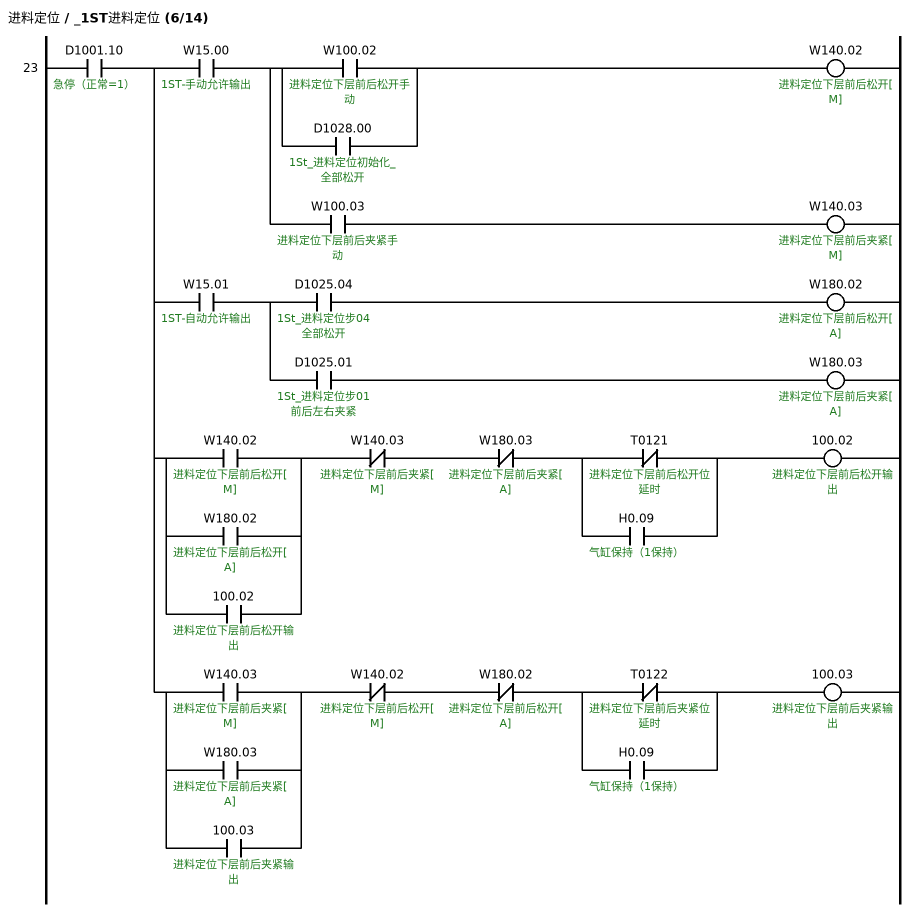
; rung 23
LD D1001.10  ; 急停（正常=1）
OUT TR0
AND W15.00  ; 1ST-手动允许输出
OUT TR1
LD W100.02  ; 进料定位下层前后松开手动
OR D1028.00  ; 1St_进料定位初始化_全部松开
ANDLD
OUT W140.02  ; 进料定位下层前后松开[M]
LD TR1
AND W100.03  ; 进料定位下层前后夹紧手动
OUT W140.03  ; 进料定位下层前后夹紧[M]
LD TR0
AND W15.01  ; 1ST-自动允许输出
OUT TR1
AND D1025.04  ; 1St_进料定位步04 全部松开
OUT W180.02  ; 进料定位下层前后松开[A]
LD TR1
AND D1025.01  ; 1St_进料定位步01 前后左右夹紧
OUT W180.03  ; 进料定位下层前后夹紧[A]
LD TR0
LD W140.02  ; 进料定位下层前后松开[M]
OR W180.02  ; 进料定位下层前后松开[A]
OR 100.02  ; 进料定位下层前后松开输出
ANDLD
ANDNOT W140.03  ; 进料定位下层前后夹紧[M]
ANDNOT W180.03  ; 进料定位下层前后夹紧[A]
LDNOT T0121  ; 进料定位下层前后松开位延时
OR H0.09  ; 气缸保持（1保持）
ANDLD
OUT 100.02  ; 进料定位下层前后松开输出
LD TR0
LD W140.03  ; 进料定位下层前后夹紧[M]
OR W180.03  ; 进料定位下层前后夹紧[A]
OR 100.03  ; 进料定位下层前后夹紧输出
ANDLD
ANDNOT W140.02  ; 进料定位下层前后松开[M]
ANDNOT W180.02  ; 进料定位下层前后松开[A]
LDNOT T0122  ; 进料定位下层前后夹紧位延时
OR H0.09  ; 气缸保持（1保持）
ANDLD
OUT 100.03  ; 进料定位下层前后夹紧输出

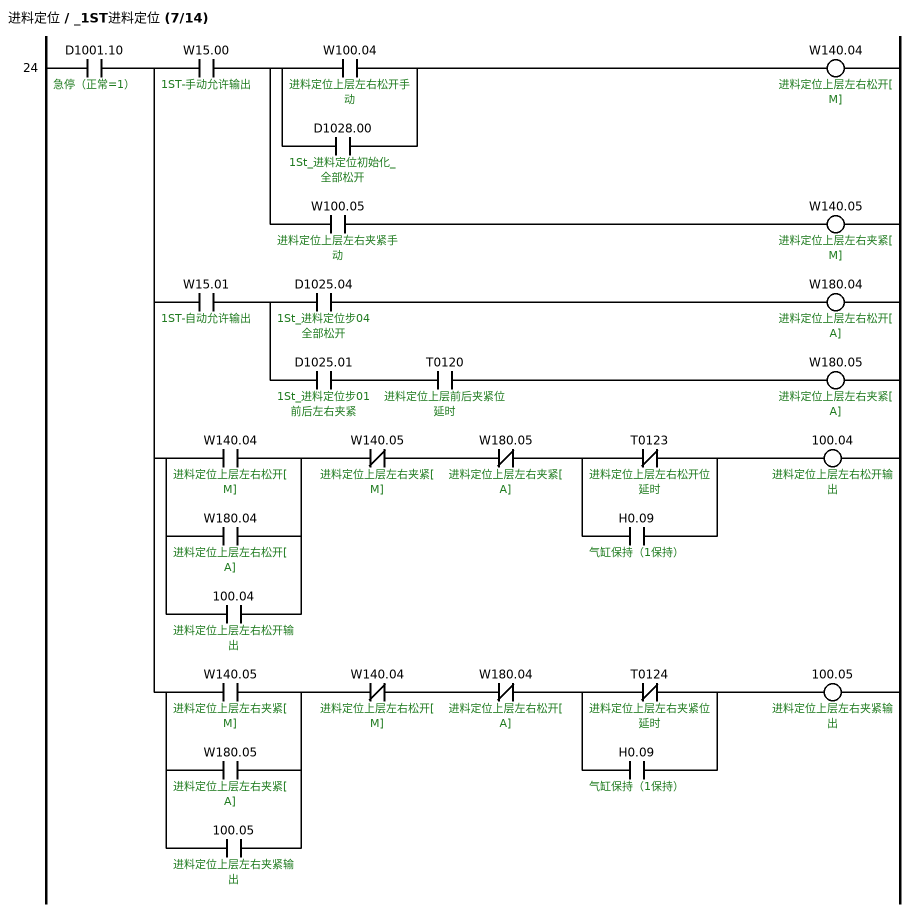
; rung 24
LD D1001.10  ; 急停（正常=1）
OUT TR0
AND W15.00  ; 1ST-手动允许输出
OUT TR1
LD W100.04  ; 进料定位上层左右松开手动
OR D1028.00  ; 1St_进料定位初始化_全部松开
ANDLD
OUT W140.04  ; 进料定位上层左右松开[M]
LD TR1
AND W100.05  ; 进料定位上层左右夹紧手动
OUT W140.05  ; 进料定位上层左右夹紧[M]
LD TR0
AND W15.01  ; 1ST-自动允许输出
OUT TR1
AND D1025.04  ; 1St_进料定位步04 全部松开
OUT W180.04  ; 进料定位上层左右松开[A]
LD TR1
AND D1025.01  ; 1St_进料定位步01 前后左右夹紧
AND T0120  ; 进料定位上层前后夹紧位延时
OUT W180.05  ; 进料定位上层左右夹紧[A]
LD TR0
LD W140.04  ; 进料定位上层左右松开[M]
OR W180.04  ; 进料定位上层左右松开[A]
OR 100.04  ; 进料定位上层左右松开输出
ANDLD
ANDNOT W140.05  ; 进料定位上层左右夹紧[M]
ANDNOT W180.05  ; 进料定位上层左右夹紧[A]
LDNOT T0123  ; 进料定位上层左右松开位延时
OR H0.09  ; 气缸保持（1保持）
ANDLD
OUT 100.04  ; 进料定位上层左右松开输出
LD TR0
LD W140.05  ; 进料定位上层左右夹紧[M]
OR W180.05  ; 进料定位上层左右夹紧[A]
OR 100.05  ; 进料定位上层左右夹紧输出
ANDLD
ANDNOT W140.04  ; 进料定位上层左右松开[M]
ANDNOT W180.04  ; 进料定位上层左右松开[A]
LDNOT T0124  ; 进料定位上层左右夹紧位延时
OR H0.09  ; 气缸保持（1保持）
ANDLD
OUT 100.05  ; 进料定位上层左右夹紧输出

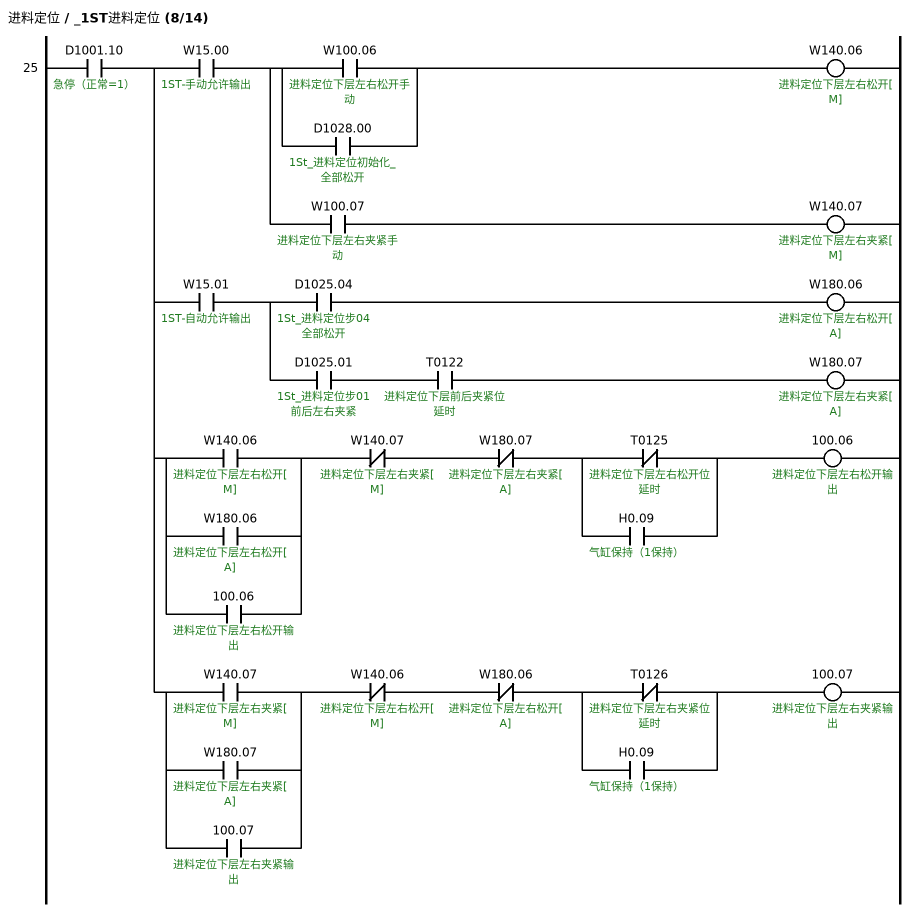
; rung 25
LD D1001.10  ; 急停（正常=1）
OUT TR0
AND W15.00  ; 1ST-手动允许输出
OUT TR1
LD W100.06  ; 进料定位下层左右松开手动
OR D1028.00  ; 1St_进料定位初始化_全部松开
ANDLD
OUT W140.06  ; 进料定位下层左右松开[M]
LD TR1
AND W100.07  ; 进料定位下层左右夹紧手动
OUT W140.07  ; 进料定位下层左右夹紧[M]
LD TR0
AND W15.01  ; 1ST-自动允许输出
OUT TR1
AND D1025.04  ; 1St_进料定位步04 全部松开
OUT W180.06  ; 进料定位下层左右松开[A]
LD TR1
AND D1025.01  ; 1St_进料定位步01 前后左右夹紧
AND T0122  ; 进料定位下层前后夹紧位延时
OUT W180.07  ; 进料定位下层左右夹紧[A]
LD TR0
LD W140.06  ; 进料定位下层左右松开[M]
OR W180.06  ; 进料定位下层左右松开[A]
OR 100.06  ; 进料定位下层左右松开输出
ANDLD
ANDNOT W140.07  ; 进料定位下层左右夹紧[M]
ANDNOT W180.07  ; 进料定位下层左右夹紧[A]
LDNOT T0125  ; 进料定位下层左右松开位延时
OR H0.09  ; 气缸保持（1保持）
ANDLD
OUT 100.06  ; 进料定位下层左右松开输出
LD TR0
LD W140.07  ; 进料定位下层左右夹紧[M]
OR W180.07  ; 进料定位下层左右夹紧[A]
OR 100.07  ; 进料定位下层左右夹紧输出
ANDLD
ANDNOT W140.06  ; 进料定位下层左右松开[M]
ANDNOT W180.06  ; 进料定位下层左右松开[A]
LDNOT T0126  ; 进料定位下层左右夹紧位延时
OR H0.09  ; 气缸保持（1保持）
ANDLD
OUT 100.07  ; 进料定位下层左右夹紧输出

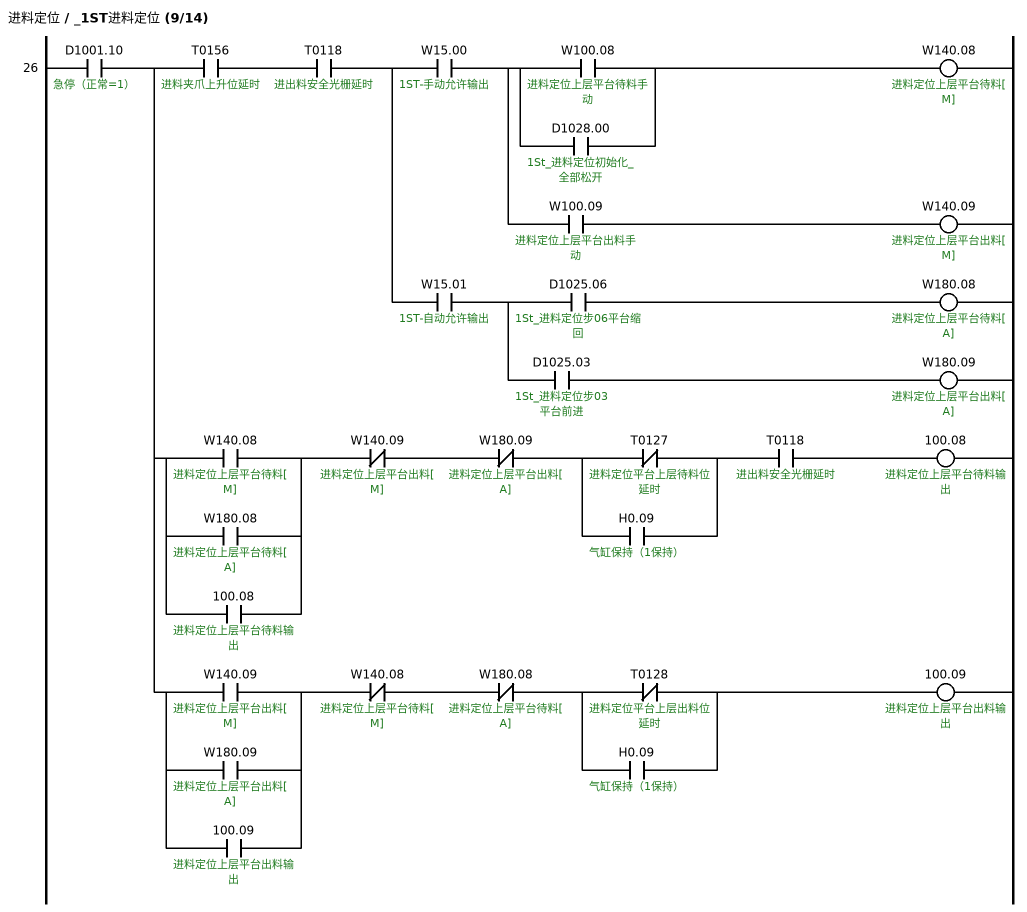
; rung 26
LD D1001.10  ; 急停（正常=1）
OUT TR0
AND T0156  ; 进料夹爪上升位延时
AND T0118  ; 进出料安全光栅延时
OUT TR1
AND W15.00  ; 1ST-手动允许输出
OUT TR2
LD W100.08  ; 进料定位上层平台待料手动
OR D1028.00  ; 1St_进料定位初始化_全部松开
ANDLD
OUT W140.08  ; 进料定位上层平台待料[M]
LD TR2
AND W100.09  ; 进料定位上层平台出料手动
OUT W140.09  ; 进料定位上层平台出料[M]
LD TR1
AND W15.01  ; 1ST-自动允许输出
OUT TR1
AND D1025.06  ; 1St_进料定位步06平台缩回
OUT W180.08  ; 进料定位上层平台待料[A]
LD TR1
AND D1025.03  ; 1St_进料定位步03 平台前进
OUT W180.09  ; 进料定位上层平台出料[A]
LD TR0
LD W140.08  ; 进料定位上层平台待料[M]
OR W180.08  ; 进料定位上层平台待料[A]
OR 100.08  ; 进料定位上层平台待料输出
ANDLD
ANDNOT W140.09  ; 进料定位上层平台出料[M]
ANDNOT W180.09  ; 进料定位上层平台出料[A]
LDNOT T0127  ; 进料定位平台上层待料位延时
OR H0.09  ; 气缸保持（1保持）
ANDLD
AND T0118  ; 进出料安全光栅延时
OUT 100.08  ; 进料定位上层平台待料输出
LD TR0
LD W140.09  ; 进料定位上层平台出料[M]
OR W180.09  ; 进料定位上层平台出料[A]
OR 100.09  ; 进料定位上层平台出料输出
ANDLD
ANDNOT W140.08  ; 进料定位上层平台待料[M]
ANDNOT W180.08  ; 进料定位上层平台待料[A]
LDNOT T0128  ; 进料定位平台上层出料位延时
OR H0.09  ; 气缸保持（1保持）
ANDLD
OUT 100.09  ; 进料定位上层平台出料输出

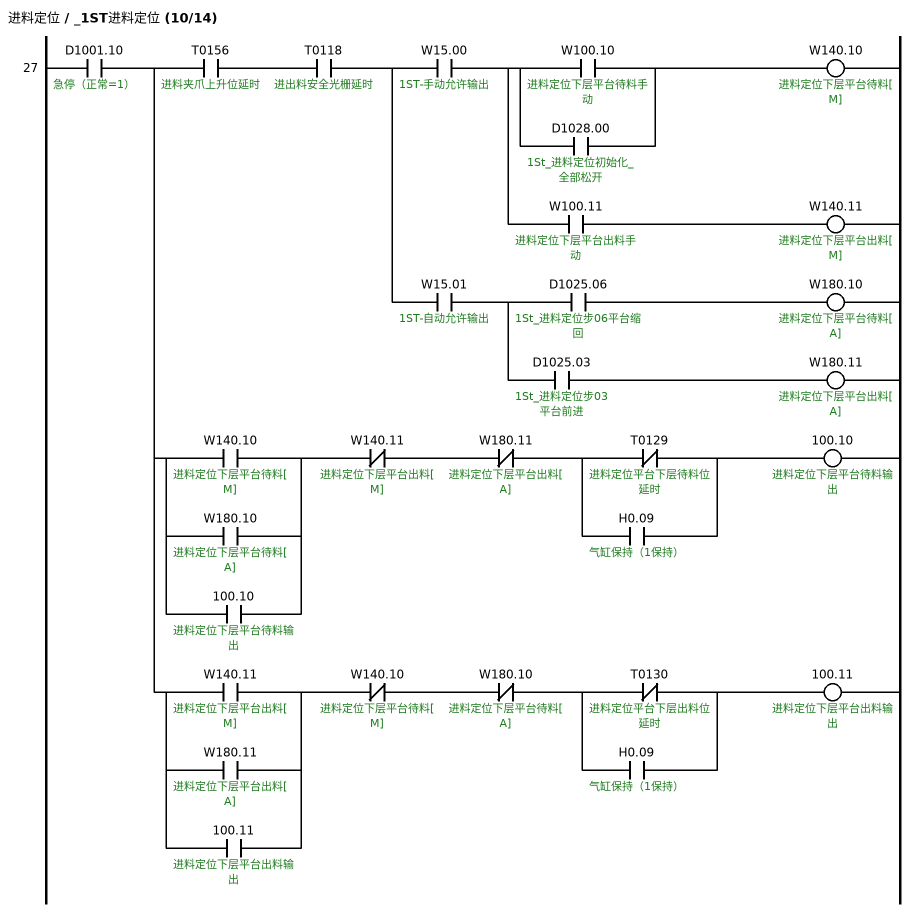
; rung 27
LD D1001.10  ; 急停（正常=1）
OUT TR0
AND T0156  ; 进料夹爪上升位延时
AND T0118  ; 进出料安全光栅延时
OUT TR1
AND W15.00  ; 1ST-手动允许输出
OUT TR2
LD W100.10  ; 进料定位下层平台待料手动
OR D1028.00  ; 1St_进料定位初始化_全部松开
ANDLD
OUT W140.10  ; 进料定位下层平台待料[M]
LD TR2
AND W100.11  ; 进料定位下层平台出料手动
OUT W140.11  ; 进料定位下层平台出料[M]
LD TR1
AND W15.01  ; 1ST-自动允许输出
OUT TR1
AND D1025.06  ; 1St_进料定位步06平台缩回
OUT W180.10  ; 进料定位下层平台待料[A]
LD TR1
AND D1025.03  ; 1St_进料定位步03 平台前进
OUT W180.11  ; 进料定位下层平台出料[A]
LD TR0
LD W140.10  ; 进料定位下层平台待料[M]
OR W180.10  ; 进料定位下层平台待料[A]
OR 100.10  ; 进料定位下层平台待料输出
ANDLD
ANDNOT W140.11  ; 进料定位下层平台出料[M]
ANDNOT W180.11  ; 进料定位下层平台出料[A]
LDNOT T0129  ; 进料定位平台下层待料位延时
OR H0.09  ; 气缸保持（1保持）
ANDLD
OUT 100.10  ; 进料定位下层平台待料输出
LD TR0
LD W140.11  ; 进料定位下层平台出料[M]
OR W180.11  ; 进料定位下层平台出料[A]
OR 100.11  ; 进料定位下层平台出料输出
ANDLD
ANDNOT W140.10  ; 进料定位下层平台待料[M]
ANDNOT W180.10  ; 进料定位下层平台待料[A]
LDNOT T0130  ; 进料定位平台下层出料位延时
OR H0.09  ; 气缸保持（1保持）
ANDLD
OUT 100.11  ; 进料定位下层平台出料输出

